RoboDK station: robodk_to_mujoco.rdk

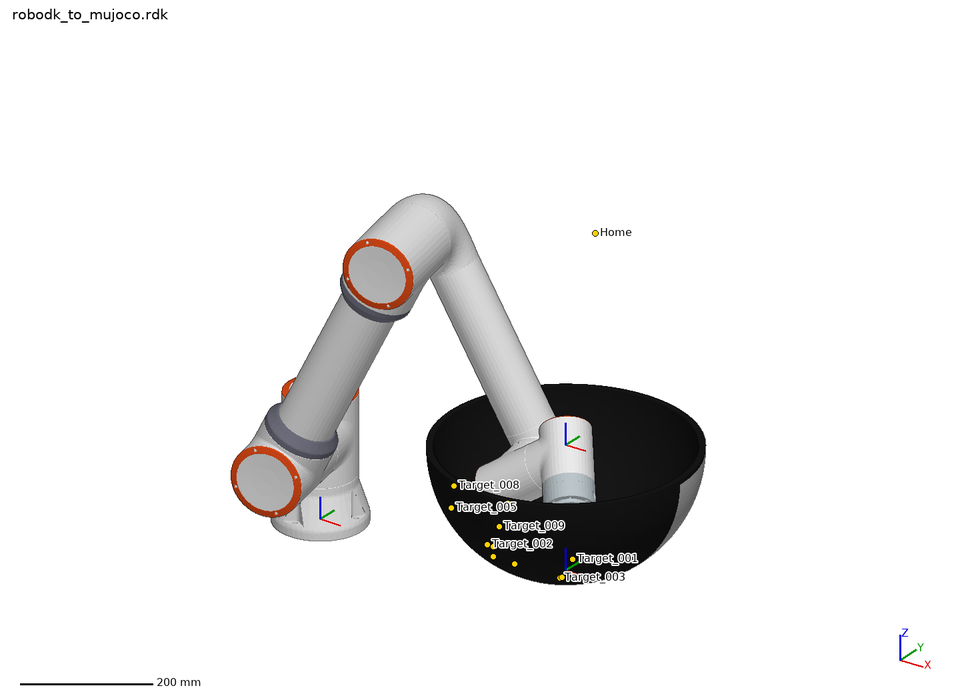
[picture v0: the station drawn from its stored meshes, robots at their saved joint values, targets as dots, program paths as lines]
Station robodk_to_mujoco (saved by RoboDK 6.0.4). Poses are relative to the parent item; angles as X-Y-Z fixed-axis rotations.
  - frame Frame 2 at (450, 0, 40) mm
    - object hemisphere at (0, 0, 0) mm, size 420 x 420 x 210 mm, geometry from hemisphere.stl
    - target Home (Cartesian target) at (125, -102, 639) mm, rotated rx -90 ry 0 rz -90 deg; joints [0, -90, -90, 0, 90, 0] of FAIRINO FR5
  - frame Hemisphere at (450, 0, 250) mm
    - target Target_001 (Cartesian target) at (103.98, -130.98, -109.55) mm, rotated rx -150.15 ry -49.64 rz -88.7 deg; joints [11.01, -115.657, -126.913, 6.584, 42.663, -19.616] of FAIRINO FR5
    - target Target_002 (Cartesian target) at (-27.22, -165.76, -108.46) mm, rotated rx 170.32 ry -55.26 rz -87.22 deg; joints [10.814, -99.215, -126.629, -70.629, 38.869, 25.952] of FAIRINO FR5
    - target Target_003 (Cartesian target) at (49.52, -85.58, -173.76) mm, rotated rx -169.33 ry -27.76 rz -82.44 deg; joints [11.892, -109.143, -129.715, -21.352, 61.937, -0.761] of FAIRINO FR5
    - target Target_004 (Cartesian target) at (-52.82, -113.56, -155.83) mm, rotated rx 159.03 ry -32.8 rz -80.27 deg; joints [11.572, -100.104, -127.366, -68.009, 60.393, 14.919] of FAIRINO FR5
    - target Target_005 (Cartesian target) at (-136.42, -105.47, -101.16) mm, rotated rx 129.4 ry -35.1 rz -77 deg; joints [12.238, -97.635, -120.965, -107.332, 67.961, 28.053] of FAIRINO FR5
    - target Target_006 (Cartesian target) at (-87.11, -65.19, -167.75) mm, rotated rx 153.07 ry -18.88 rz -87.14 deg; joints [12.149, -99.358, -126.978, -73.988, 77.779, 17.168] of FAIRINO FR5
    - target Target_007 (Cartesian target) at (-42.61, -73.24, -181.14) mm, rotated rx 166.82 ry -19.98 rz -86.86 deg; joints [11.803, -101.566, -129.071, -56.123, 72.868, 13.541] of FAIRINO FR5
    - target Target_008 (Cartesian target) at (-167.97, -52.04, -95.08) mm, rotated rx 120.74 ry -21.46 rz -84.25 deg; joints [13.234, -98.115, -119.768, -113.628, 85.788, 22.298] of FAIRINO FR5
    - target Target_009 (Cartesian target) at (-113.79, -12.21, -163.93) mm, rotated rx 145.41 ry -7.9 rz -94.34 deg; joints [13.464, -98.923, -126.265, -80.011, 93.775, 19.074] of FAIRINO FR5
    - target Target_010 (Cartesian target) at (-130.39, 34.76, -147.56) mm, rotated rx 138.81 ry 1.53 rz -102.65 deg; joints [14.271, -97.609, -126.165, -83.767, 108.427, 20.04] of FAIRINO FR5
    - target Target_011 (Cartesian target) at (32.97, -56.8, -188.88) mm, rotated rx -173.19 ry -16.73 rz -82.94 deg; joints [11.888, -108.019, -129.691, -26.64, 72.85, 2.973] of FAIRINO FR5
  - frame FAIRINO FR5 Base at (0, 0, 0) mm
    - robot FAIRINO FR5: 6 axes
        modified DH rows (alpha deg, a mm, theta deg, d mm): 0, 0, 0, 152; 90, 0, 180, 0; 0, 425, 0, 0; 0, 395, 0, 102; -90, 0, 0, 102; 90, 0, 180, 100
        joint limits [-175, -265, -160, -265, -175, -175] to [175, 85, 160, 85, 175, 175]; home [0, -90, -90, 0, 90, 0]; saved at [11.01, -115.657, -126.913, 6.584, 42.663, -19.616]
      - tool Tool 1, TCP at (0, 0, 80) mm
